// TIA Portal V19 export
FUNCTION "PitTable1_CALL" : Void   // FC183, LAD
TITLE = CALL PIT TABLE LOOP @ ENTRY OF ROLLFORMER (DOWN = REST / UP = WORK)
// stored: SetENOAutomatically false
BEGIN

REGION Network 1: Data In - PB
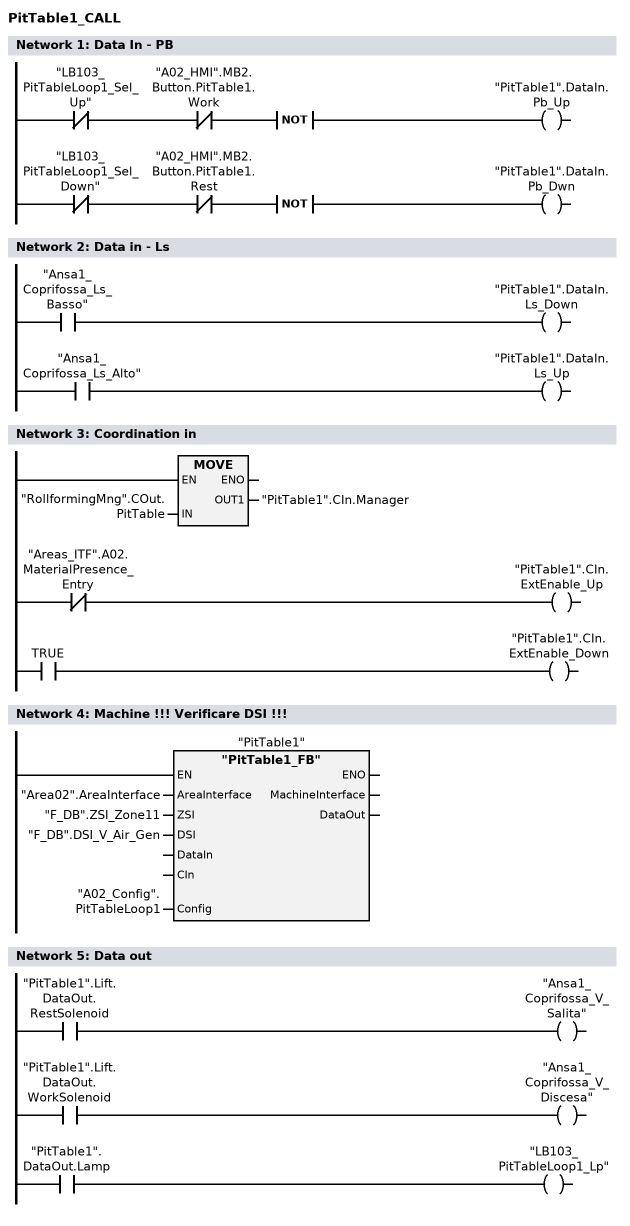
   RUNG wire#powerrail
      I_Contact( "LB103_PitTableLoop1_Sel_Up" )
      I_Contact( "A02_HMI".MB2.Button.PitTable1.Work )
      Not()
      Coil( "PitTable1".DataIn.Pb_Up )
   END_RUNG
   RUNG wire#powerrail
      I_Contact( "LB103_PitTableLoop1_Sel_Down" )
      I_Contact( "A02_HMI".MB2.Button.PitTable1.Rest )
      Not()
      Coil( "PitTable1".DataIn.Pb_Dwn )
   END_RUNG
   // the same network as SCL:
   "PitTable1".DataIn.Pb_Up := NOT (NOT "LB103_PitTableLoop1_Sel_Up" AND NOT "A02_HMI".MB2.Button.PitTable1.Work);
   "PitTable1".DataIn.Pb_Dwn := NOT (NOT "LB103_PitTableLoop1_Sel_Down" AND NOT "A02_HMI".MB2.Button.PitTable1.Rest);
END_REGION

REGION Network 2: Data in - Ls
   RUNG wire#powerrail
      Contact( "Ansa1_Coprifossa_Ls_Basso" )
      Coil( "PitTable1".DataIn.Ls_Down )
   END_RUNG
   RUNG wire#powerrail
      Contact( "Ansa1_Coprifossa_Ls_Alto" )
      Coil( "PitTable1".DataIn.Ls_Up )
   END_RUNG
   // the same network as SCL:
   "PitTable1".DataIn.Ls_Down := "Ansa1_Coprifossa_Ls_Basso";
   "PitTable1".DataIn.Ls_Up := "Ansa1_Coprifossa_Ls_Alto";
END_REGION

REGION Network 3: Coordination in
   RUNG wire#powerrail
      { S7_GenerateENO := "TRUE" } Move(in := "RollformingMng".COut.PitTable, out1 => "PitTable1".CIn.Manager)
   END_RUNG
   RUNG wire#powerrail
      I_Contact( "Areas_ITF".A02.MaterialPresence_Entry )
      Coil( "PitTable1".CIn.ExtEnable_Up )
   END_RUNG
   RUNG wire#powerrail
      Contact( TRUE )
      Coil( "PitTable1".CIn.ExtEnable_Down )
   END_RUNG
   // the same network as SCL:
   "PitTable1".CIn.Manager := "RollformingMng".COut.PitTable;
   "PitTable1".CIn.ExtEnable_Up := NOT "Areas_ITF".A02.MaterialPresence_Entry;
   "PitTable1".CIn.ExtEnable_Down := TRUE;
END_REGION

REGION Network 4: Machine !!! Verificare DSI !!!
   RUNG wire#powerrail
      "PitTable1"(AreaInterface := "Area02".AreaInterface, ZSI := "F_DB".ZSI_Zone11, DSI := "F_DB".DSI_V_Air_Gen, DataIn :=, CIn :=, Config := "A02_Config".PitTableLoop1, MachineInterface =>, DataOut =>)
   END_RUNG
   // the same network as SCL:
   "PitTable1"(AreaInterface := "Area02".AreaInterface,   // "PitTable1_FB"
               ZSI := "F_DB".ZSI_Zone11,
               DSI := "F_DB".DSI_V_Air_Gen,
               Config := "A02_Config".PitTableLoop1);
END_REGION

REGION Network 5: Data out
   RUNG wire#powerrail
      Contact( "PitTable1".Lift.DataOut.RestSolenoid )
      Coil( "Ansa1_Coprifossa_V_Salita" )
   END_RUNG
   RUNG wire#powerrail
      Contact( "PitTable1".Lift.DataOut.WorkSolenoid )
      Coil( "Ansa1_Coprifossa_V_Discesa" )
   END_RUNG
   RUNG wire#powerrail
      Contact( "PitTable1".DataOut.Lamp )
      Coil( "LB103_PitTableLoop1_Lp" )
   END_RUNG
   // the same network as SCL:
   "Ansa1_Coprifossa_V_Salita" := "PitTable1".Lift.DataOut.RestSolenoid;
   "Ansa1_Coprifossa_V_Discesa" := "PitTable1".Lift.DataOut.WorkSolenoid;
   "LB103_PitTableLoop1_Lp" := "PitTable1".DataOut.Lamp;
END_REGION

REGION Network 6: >
END_REGION

REGION Network 7: >
END_REGION

REGION Network 8: >
END_REGION
END_FUNCTION
